(* PLC project Untitled1, Eclipse Foundation CIF to Structured Text 0.0 *)
(* stored: creationDateTime 1970-01-01T00:00:00Z *)

TYPE STATE : STRUCT
  curTime : LREAL;
  cvar_c AT %Q* : LREAL;
  dvar_M_aut_r AT %Q* : LREAL;
  dvar_M_aut_b AT %Q* : BOOL;
  dvar_M_aut_i AT %Q* : DINT;
  dvar_M_aut_tii AT %Q* : TupleStruct_1;
  dvar_M_aut_i2 AT %Q* : DINT;
  dvar_M_aut_i3 AT %Q* : DINT;
  dvar_M_aut AT %Q* : enum_E;
END_STRUCT;
END_TYPE

TYPE enum_E : (elit_l1, elit_l2);
END_TYPE

TYPE TupleStruct_1 : STRUCT
  field0 : DINT;
  field1 : DINT;
END_STRUCT;
END_TYPE

TYPE TupleStruct_2 : STRUCT
  field0 : LREAL;
  field1 : DINT;
END_STRUCT;
END_TYPE

FUNCTION derivcvar_c : LREAL
  VAR_INPUT
    state : STATE;
  END_VAR

            derivcvar_c := state.cvar_c;
          
END_FUNCTION

FUNCTION alg_a : LREAL
  VAR_INPUT
    state : STATE;
  END_VAR

            alg_a := (state.cvar_c) + (derivcvar_c(state));
          
END_FUNCTION

FUNCTION ifExprFunc1 : BOOL
  VAR_INPUT
    dummy : INT;
  END_VAR

            IF (func_f1(TRUE)) THEN
    ifExprFunc1 := TRUE;
ELSE
    ifExprFunc1 := TRUE;
END_IF;
          
END_FUNCTION

FUNCTION func_f1 : BOOL
  VAR_INPUT
    farg_f1_p : BOOL;
  END_VAR

            func_f1 := (farg_f1_p) AND (ifExprFunc1(0));
RETURN;
          
END_FUNCTION

FUNCTION ifExprFunc2 : BOOL
  VAR_INPUT
    farg_f2_p : BOOL;
  END_VAR

            IF (farg_f2_p) THEN
    ifExprFunc2 := TRUE;
ELSE
    ifExprFunc2 := TRUE;
END_IF;
          
END_FUNCTION

FUNCTION func_f2 : BOOL
  VAR_INPUT
    farg_f2_p : BOOL;
  END_VAR

            func_f2 := ifExprFunc2(farg_f2_p);
RETURN;
          
END_FUNCTION

FUNCTION makeTupleStruct_1 : TupleStruct_1
  VAR_INPUT
    field0 : DINT;
    field1 : DINT;
  END_VAR
  VAR
    rslt : TupleStruct_1;
  END_VAR

            rslt.field0 := field0;
rslt.field1 := field1;
makeTupleStruct_1 := rslt;
          
END_FUNCTION

FUNCTION proj0_TupleStruct_1 : DINT
  VAR_INPUT
    tuple : TupleStruct_1;
  END_VAR

            proj0_TupleStruct_1 := tuple.field0;
          
END_FUNCTION

FUNCTION proj1_TupleStruct_1 : DINT
  VAR_INPUT
    tuple : TupleStruct_1;
  END_VAR

            proj1_TupleStruct_1 := tuple.field1;
          
END_FUNCTION

FUNCTION ifExprFunc3 : BOOL
  VAR_INPUT
    state : STATE;
  END_VAR

            IF (state.dvar_M_aut_b) THEN
    ifExprFunc3 := state.dvar_M_aut_b;
ELSE
    ifExprFunc3 := state.dvar_M_aut_b;
END_IF;
          
END_FUNCTION

FUNCTION makeTupleStruct_2 : TupleStruct_2
  VAR_INPUT
    field0 : LREAL;
    field1 : DINT;
  END_VAR
  VAR
    rslt : TupleStruct_2;
  END_VAR

            rslt.field0 := field0;
rslt.field1 := field1;
makeTupleStruct_2 := rslt;
          
END_FUNCTION

FUNCTION proj0_TupleStruct_2 : LREAL
  VAR_INPUT
    tuple : TupleStruct_2;
  END_VAR

            proj0_TupleStruct_2 := tuple.field0;
          
END_FUNCTION

FUNCTION proj1_TupleStruct_2 : DINT
  VAR_INPUT
    tuple : TupleStruct_2;
  END_VAR

            proj1_TupleStruct_2 := tuple.field1;
          
END_FUNCTION

PROGRAM MAIN
  VAR_OUTPUT
    timerValue0 : TIME;
    timerValue1 : TIME;
  END_VAR
  VAR
    cnt : LINT;
    first : BOOL := TRUE;
    curTimerValue : TIME;
    state0 : STATE;
    curTime : LREAL;
    loopsKilled : LINT;
  END_VAR
  VAR_TEMP
    lastTimerValue : TIME;
    curDeltaTime : TIME;
    curDeltaSecs : LREAL;
    state1 : STATE;
    progress : BOOL;
    loopCount : INT;
    b1 : BOOL;
    b2 : BOOL;
  END_VAR

            
// Handle 'time' and cycle time.
cnt := cnt + 1;

timer0(IN := curTimer = 0, PT := T#1D);
timer1(IN := curTimer = 1, PT := T#1D);
timerValue0 := timer0.ET;
timerValue1 := timer1.ET;

lastTimerValue := curTimerValue;
IF curTimer = 0 THEN
    curTimerValue := timerValue0;
ELSE
    curTimerValue := timerValue1;
END_IF;
curDeltaTime := curTimerValue - lastTimerValue;
curDeltaSecs := TIME_TO_LREAL(curDeltaTime) / 1000;
curTime := curTime + curDeltaSecs;

IF cnt MOD 10 = 0 THEN
    curTimer := 1 - curTimer;
    curTimerValue := T#0S;
    timer0(IN := curTimer = 0, PT := T#1D);
    timer1(IN := curTimer = 1, PT := T#1D);
    timerValue0 := timer0.ET;
    timerValue1 := timer1.ET;
END_IF;

IF first THEN
    first := FALSE;

    // Initialize state variables for initial state.
    state0.cvar_c := 0.0;
    state0.dvar_M_aut_r := 0.0;
    state0.dvar_M_aut_b := FALSE;
    state0.dvar_M_aut_i := 0;
    state0.dvar_M_aut_tii := makeTupleStruct_1(0, 0);
    state0.dvar_M_aut_i2 := 1;
    state0.dvar_M_aut_i3 := 1;
    state0.dvar_M_aut := elit_l1;
ELSE
    // Update continuous variables for time delay.
    state1.cvar_c := state0.cvar_c + curDeltaSecs * derivcvar_c(state0);

    state0.curTime := curTime;
    state0.cvar_c := state1.cvar_c;
END_IF;

// Event loop.
WHILE TRUE DO
    progress := FALSE;

    // Event "M.aut_e".
    IF NOT progress THEN
        b1 := (state0.dvar_M_aut) = (elit_l1);
        IF b1 THEN
            b2 := state0.dvar_M_aut_b;
            b2 := b2 OR (state0.dvar_M_aut_b);
            b2 := b2 OR (state0.dvar_M_aut_b);
            b1 := b1 AND (b2);
        END_IF;
        IF b1 THEN
            progress := TRUE;
            state1 := state0;


            state0 := state1;
        END_IF;
    END_IF;

    // Event "tau".
    IF NOT progress THEN
        IF (state0.dvar_M_aut) = (elit_l1) THEN
            progress := TRUE;
            state1 := state0;

            state1.dvar_M_aut_r := ivar_inp;

            state0 := state1;
        END_IF;
    END_IF;

    // Event "tau".
    IF NOT progress THEN
        IF (state0.dvar_M_aut) = (elit_l1) THEN
            progress := TRUE;
            state1 := state0;

            state1.dvar_M_aut_r := ((alg_a(state0)) + (state0.cvar_c)) + (derivcvar_c(state0));
            state1.dvar_M_aut := elit_l2;

            state0 := state1;
        END_IF;
    END_IF;

    // Event "tau".
    IF NOT progress THEN
        IF (state0.dvar_M_aut) = (elit_l1) THEN
            progress := TRUE;
            state1 := state0;

            state1.dvar_M_aut_r := DINT_TO_LREAL(state0.dvar_M_aut_i);

            state0 := state1;
        END_IF;
    END_IF;

    // Event "tau".
    IF NOT progress THEN
        IF (state0.dvar_M_aut) = (elit_l1) THEN
            progress := TRUE;
            state1 := state0;

            state1.dvar_M_aut_b := NOT(state0.dvar_M_aut_b);

            state0 := state1;
        END_IF;
    END_IF;

    // Event "tau".
    IF NOT progress THEN
        IF (state0.dvar_M_aut) = (elit_l1) THEN
            progress := TRUE;
            state1 := state0;

            state1.dvar_M_aut_b := NOT(state0.dvar_M_aut_b) OR (state0.dvar_M_aut_b);

            state0 := state1;
        END_IF;
    END_IF;

    // Event "tau".
    IF NOT progress THEN
        IF (state0.dvar_M_aut) = (elit_l1) THEN
            progress := TRUE;
            state1 := state0;

            state1.dvar_M_aut_r := DINT_TO_LREAL(state0.dvar_M_aut_i) / (state0.dvar_M_aut_i);

            state0 := state1;
        END_IF;
    END_IF;

    // Event "tau".
    IF NOT progress THEN
        IF (state0.dvar_M_aut) = (elit_l1) THEN
            progress := TRUE;
            state1 := state0;

            state1.dvar_M_aut_b := func_f1(state0.dvar_M_aut_b);

            state0 := state1;
        END_IF;
    END_IF;

    // Event "tau".
    IF NOT progress THEN
        IF (state0.dvar_M_aut) = (elit_l1) THEN
            progress := TRUE;
            state1 := state0;

            state1.dvar_M_aut_b := func_f2(state0.dvar_M_aut_b);

            state0 := state1;
        END_IF;
    END_IF;

    // Event "tau".
    IF NOT progress THEN
        IF (state0.dvar_M_aut) = (elit_l1) THEN
            progress := TRUE;
            state1 := state0;

            state1.dvar_M_aut_b := ifExprFunc3(state0);

            state0 := state1;
        END_IF;
    END_IF;

    // Event "tau".
    IF NOT progress THEN
        IF (state0.dvar_M_aut) = (elit_l1) THEN
            progress := TRUE;
            state1 := state0;

            state1.dvar_M_aut_i := proj0_TupleStruct_1(state0.dvar_M_aut_tii);

            state0 := state1;
        END_IF;
    END_IF;

    // Event "tau".
    IF NOT progress THEN
        IF (state0.dvar_M_aut) = (elit_l1) THEN
            progress := TRUE;
            state1 := state0;

            state1.dvar_M_aut_r := ABS(state0.dvar_M_aut_r);

            state0 := state1;
        END_IF;
    END_IF;

    // Event "tau".
    IF NOT progress THEN
        IF (state0.dvar_M_aut) = (elit_l1) THEN
            progress := TRUE;
            state1 := state0;

            state1.dvar_M_aut_r := EXPT(state0.dvar_M_aut_r, 1.0/3);

            state0 := state1;
        END_IF;
    END_IF;

    // Event "tau".
    IF NOT progress THEN
        IF (state0.dvar_M_aut) = (elit_l1) THEN
            progress := TRUE;
            state1 := state0;

            state1.dvar_M_aut_r := EXP(state0.dvar_M_aut_r);

            state0 := state1;
        END_IF;
    END_IF;

    // Event "tau".
    IF NOT progress THEN
        IF (state0.dvar_M_aut) = (elit_l1) THEN
            progress := TRUE;
            state1 := state0;

            state1.dvar_M_aut_r := LN(state0.dvar_M_aut_r);

            state0 := state1;
        END_IF;
    END_IF;

    // Event "tau".
    IF NOT progress THEN
        IF (state0.dvar_M_aut) = (elit_l1) THEN
            progress := TRUE;
            state1 := state0;

            state1.dvar_M_aut_r := LOG(state0.dvar_M_aut_r);

            state0 := state1;
        END_IF;
    END_IF;

    // Event "tau".
    IF NOT progress THEN
        IF (state0.dvar_M_aut) = (elit_l1) THEN
            progress := TRUE;
            state1 := state0;

            state1.dvar_M_aut_i := MIN(state0.dvar_M_aut_i, state0.dvar_M_aut_i);

            state0 := state1;
        END_IF;
    END_IF;

    // Event "tau".
    IF NOT progress THEN
        IF (state0.dvar_M_aut) = (elit_l1) THEN
            progress := TRUE;
            state1 := state0;

            state1.dvar_M_aut_r := MIN(DINT_TO_LREAL(state0.dvar_M_aut_i), state0.dvar_M_aut_r);

            state0 := state1;
        END_IF;
    END_IF;

    // Event "tau".
    IF NOT progress THEN
        IF (state0.dvar_M_aut) = (elit_l1) THEN
            progress := TRUE;
            state1 := state0;

            state1.dvar_M_aut_r := MIN(state0.dvar_M_aut_r, DINT_TO_LREAL(state0.dvar_M_aut_i));

            state0 := state1;
        END_IF;
    END_IF;

    // Event "tau".
    IF NOT progress THEN
        IF (state0.dvar_M_aut) = (elit_l1) THEN
            progress := TRUE;
            state1 := state0;

            state1.dvar_M_aut_r := MIN(state0.dvar_M_aut_r, state0.dvar_M_aut_r);

            state0 := state1;
        END_IF;
    END_IF;

    // Event "tau".
    IF NOT progress THEN
        IF (state0.dvar_M_aut) = (elit_l1) THEN
            progress := TRUE;
            state1 := state0;

            state1.dvar_M_aut_i := MAX(state0.dvar_M_aut_i, state0.dvar_M_aut_i);

            state0 := state1;
        END_IF;
    END_IF;

    // Event "tau".
    IF NOT progress THEN
        IF (state0.dvar_M_aut) = (elit_l1) THEN
            progress := TRUE;
            state1 := state0;

            state1.dvar_M_aut_r := MAX(DINT_TO_LREAL(state0.dvar_M_aut_i), state0.dvar_M_aut_r);

            state0 := state1;
        END_IF;
    END_IF;

    // Event "tau".
    IF NOT progress THEN
        IF (state0.dvar_M_aut) = (elit_l1) THEN
            progress := TRUE;
            state1 := state0;

            state1.dvar_M_aut_r := MAX(state0.dvar_M_aut_r, DINT_TO_LREAL(state0.dvar_M_aut_i));

            state0 := state1;
        END_IF;
    END_IF;

    // Event "tau".
    IF NOT progress THEN
        IF (state0.dvar_M_aut) = (elit_l1) THEN
            progress := TRUE;
            state1 := state0;

            state1.dvar_M_aut_r := MAX(state0.dvar_M_aut_r, state0.dvar_M_aut_r);

            state0 := state1;
        END_IF;
    END_IF;

    // Event "tau".
    IF NOT progress THEN
        IF (state0.dvar_M_aut) = (elit_l1) THEN
            progress := TRUE;
            state1 := state0;

            state1.dvar_M_aut_i := LREAL_TO_DINT(EXPT(DINT_TO_LREAL(state0.dvar_M_aut_i2), state0.dvar_M_aut_i3));

            state0 := state1;
        END_IF;
    END_IF;

    // Event "tau".
    IF NOT progress THEN
        IF (state0.dvar_M_aut) = (elit_l1) THEN
            progress := TRUE;
            state1 := state0;

            state1.dvar_M_aut_r := EXPT(state0.dvar_M_aut_i, state0.dvar_M_aut_i);

            state0 := state1;
        END_IF;
    END_IF;

    // Event "tau".
    IF NOT progress THEN
        IF (state0.dvar_M_aut) = (elit_l1) THEN
            progress := TRUE;
            state1 := state0;

            state1.dvar_M_aut_r := EXPT(DINT_TO_LREAL(state0.dvar_M_aut_i), state0.dvar_M_aut_r);

            state0 := state1;
        END_IF;
    END_IF;

    // Event "tau".
    IF NOT progress THEN
        IF (state0.dvar_M_aut) = (elit_l1) THEN
            progress := TRUE;
            state1 := state0;

            state1.dvar_M_aut_r := EXPT(state0.dvar_M_aut_r, state0.dvar_M_aut_i);

            state0 := state1;
        END_IF;
    END_IF;

    // Event "tau".
    IF NOT progress THEN
        IF (state0.dvar_M_aut) = (elit_l1) THEN
            progress := TRUE;
            state1 := state0;

            state1.dvar_M_aut_r := EXPT(state0.dvar_M_aut_r, state0.dvar_M_aut_r);

            state0 := state1;
        END_IF;
    END_IF;

    // Event "tau".
    IF NOT progress THEN
        IF (state0.dvar_M_aut) = (elit_l1) THEN
            progress := TRUE;
            state1 := state0;

            state1.dvar_M_aut_r := SQRT(state0.dvar_M_aut_r);

            state0 := state1;
        END_IF;
    END_IF;

    // Event "tau".
    IF NOT progress THEN
        IF (state0.dvar_M_aut) = (elit_l1) THEN
            progress := TRUE;
            state1 := state0;

            state1.dvar_M_aut_r := ASIN(state0.dvar_M_aut_r);

            state0 := state1;
        END_IF;
    END_IF;

    // Event "tau".
    IF NOT progress THEN
        IF (state0.dvar_M_aut) = (elit_l1) THEN
            progress := TRUE;
            state1 := state0;

            state1.dvar_M_aut_r := ACOS(state0.dvar_M_aut_r);

            state0 := state1;
        END_IF;
    END_IF;

    // Event "tau".
    IF NOT progress THEN
        IF (state0.dvar_M_aut) = (elit_l1) THEN
            progress := TRUE;
            state1 := state0;

            state1.dvar_M_aut_r := ATAN(state0.dvar_M_aut_r);

            state0 := state1;
        END_IF;
    END_IF;

    // Event "tau".
    IF NOT progress THEN
        IF (state0.dvar_M_aut) = (elit_l1) THEN
            progress := TRUE;
            state1 := state0;

            state1.dvar_M_aut_r := SIN(state0.dvar_M_aut_r);

            state0 := state1;
        END_IF;
    END_IF;

    // Event "tau".
    IF NOT progress THEN
        IF (state0.dvar_M_aut) = (elit_l1) THEN
            progress := TRUE;
            state1 := state0;

            state1.dvar_M_aut_r := COS(state0.dvar_M_aut_r);

            state0 := state1;
        END_IF;
    END_IF;

    // Event "tau".
    IF NOT progress THEN
        IF (state0.dvar_M_aut) = (elit_l1) THEN
            progress := TRUE;
            state1 := state0;

            state1.dvar_M_aut_r := TAN(state0.dvar_M_aut_r);

            state0 := state1;
        END_IF;
    END_IF;

    // Event "tau".
    IF NOT progress THEN
        IF (state0.dvar_M_aut) = (elit_l1) THEN
            progress := TRUE;
            state1 := state0;

            state1.dvar_M_aut_tii := makeTupleStruct_1(state0.dvar_M_aut_i, (state0.dvar_M_aut_i) + (1));

            state0 := state1;
        END_IF;
    END_IF;

    // Event "tau".
    IF NOT progress THEN
        IF (state0.dvar_M_aut) = (elit_l1) THEN
            progress := TRUE;
            state1 := state0;

            state1.dvar_M_aut_r := proj0_TupleStruct_2(makeTupleStruct_2((state0.dvar_M_aut_r) * (2.0), (state0.dvar_M_aut_i) + (1)));
            state1.dvar_M_aut_i := proj1_TupleStruct_2(makeTupleStruct_2((state0.dvar_M_aut_r) * (2.0), (state0.dvar_M_aut_i) + (1)));

            state0 := state1;
        END_IF;
    END_IF;

    // Done with events?
    IF NOT progress THEN
        EXIT;
    END_IF;

    // Protect against events that are always enabled.
    loopCount := loopCount + 1;
    IF loopCount >= 100 THEN
        loopsKilled := loopsKilled + 1;
        EXIT;
    END_IF;
END_WHILE;
          
END_PROGRAM

CONFIGURATION Untitled1
  RESOURCE Untitled1 ON PLC
    VAR_GLOBAL  (* INPUTS *)
      ivar_inp AT %I* : LREAL;
    END_VAR
    VAR_GLOBAL  (* TIMERS *)
      timer0 : TON;
      timer1 : TON;
      curTimer : INT := 0;
    END_VAR
    TASK PlcTask(INTERVAL := T#10ms, PRIORITY := 20);
    PROGRAM MAIN WITH PlcTask : MAIN;
  END_RESOURCE
END_CONFIGURATION
